RoboDK station: test.rdk

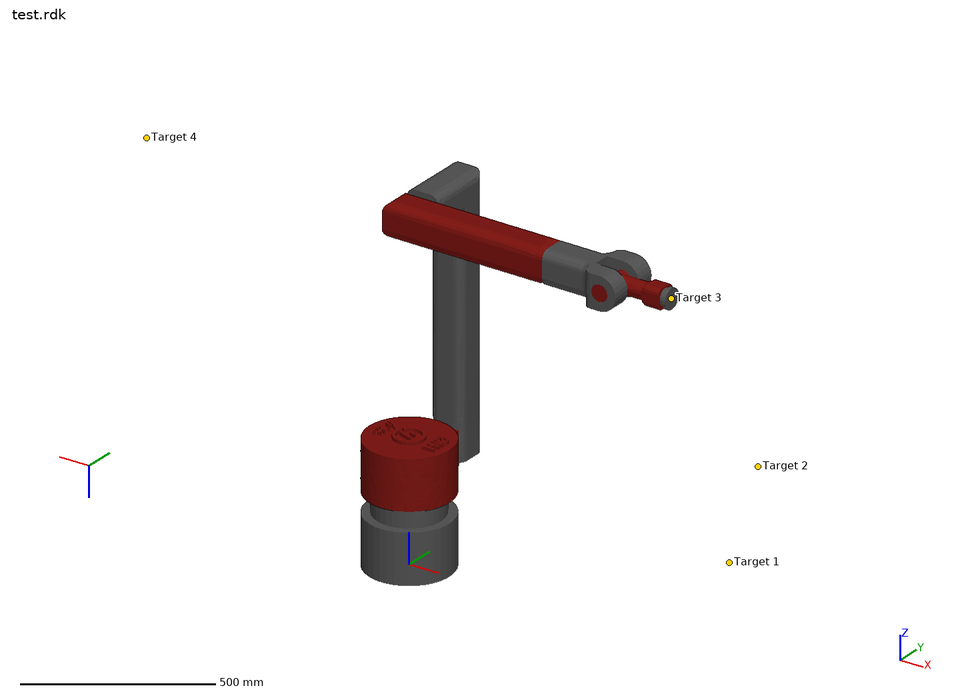
[picture v0: the station drawn from its stored meshes, robots at their saved joint values, targets as dots, program paths as lines]
Station test (saved by RoboDK 5.9.2). Poses are relative to the parent item; angles as X-Y-Z fixed-axis rotations.
  - frame My Mechanism Base at (0, 1000, 0) mm
    - robot My Mechanism: 6 axes
        modified DH rows (alpha deg, a mm, theta deg, d mm): 0, 0, 0, 285; -90, 0, -90, 0; 0, 700, -90, 0; -90, 0, 0, 650; 90, 0, 0, 0; -90, 0, 180, 170
        joint limits [-180, -90, -135, -180, -90, -180] to [180, 90, 135, 180, 90, 180]; home [0, 0, 0, 0, 0, 0]; saved at [0, 0, 90, 0, 0, 0]
    - target Target 1 (Cartesian target) at (1000, 0, 285) mm, rotated rx 180 ry 0 rz 180 deg; joints [0, 40.892, -7.349, 0, 56.457, 0] of My Mechanism
    - target Target 2 (Cartesian target) at (740, 500, 285) mm, rotated rx 180 ry 0 rz 180 deg; joints [34.046, 33.843, 5.423, 0, 50.734, 34.046] of My Mechanism
    - frame Frame 2 at (-1000, 0, 0) mm, rotated rx 180 ry 0 rz 180 deg
    - target Target 3 (Cartesian target) at (820, 0, 985) mm, rotated rx 0 ry 90 rz 0 deg; joints [0, 0, 0, 0, 0, 0] of My Mechanism
    - target Target 4 (Cartesian target) at (-820, 0, 985) mm, rotated rx 0 ry -90 rz 0 deg; joints [0, 0, -90, 0, 0, 0] of My Mechanism
  - Python program Prog1 (listed below)

--- Python program Prog1 ---
from time import sleep
from robodk.robolink import Robolink, ITEM_TYPE_TARGET, ITEM_TYPE_FRAME
RDK = Robolink()
from robot_communication import RobotSerial

robot = RobotSerial('COM5')

t1 = RDK.Item('Target 1', ITEM_TYPE_TARGET)
t2 = RDK.Item('Target 2', ITEM_TYPE_TARGET)
t3 = RDK.Item('Target 3', ITEM_TYPE_TARGET)
t4 = RDK.Item('Target 4', ITEM_TYPE_TARGET)

f2 = RDK.Item('Frame 2', ITEM_TYPE_FRAME)


robot.MoveJ(t3)

print("")
sleep(0.5)

robot.home()
"""
robot.setDO(1)
print("")
sleep(0.5)

#robot.MoveJ(t4)
robot.setDO(0)
"""
